FUNCTION_BLOCK Gerador_HMI (* HMI Gerador AGC150 - 74 vars + 33 HAB equipamentos *)
  (* Standard: 61499-2 *)
  (* Version 7.0, 13/05/2026, Claude *)
  PACKAGE Hidryco.HidrycoLib;
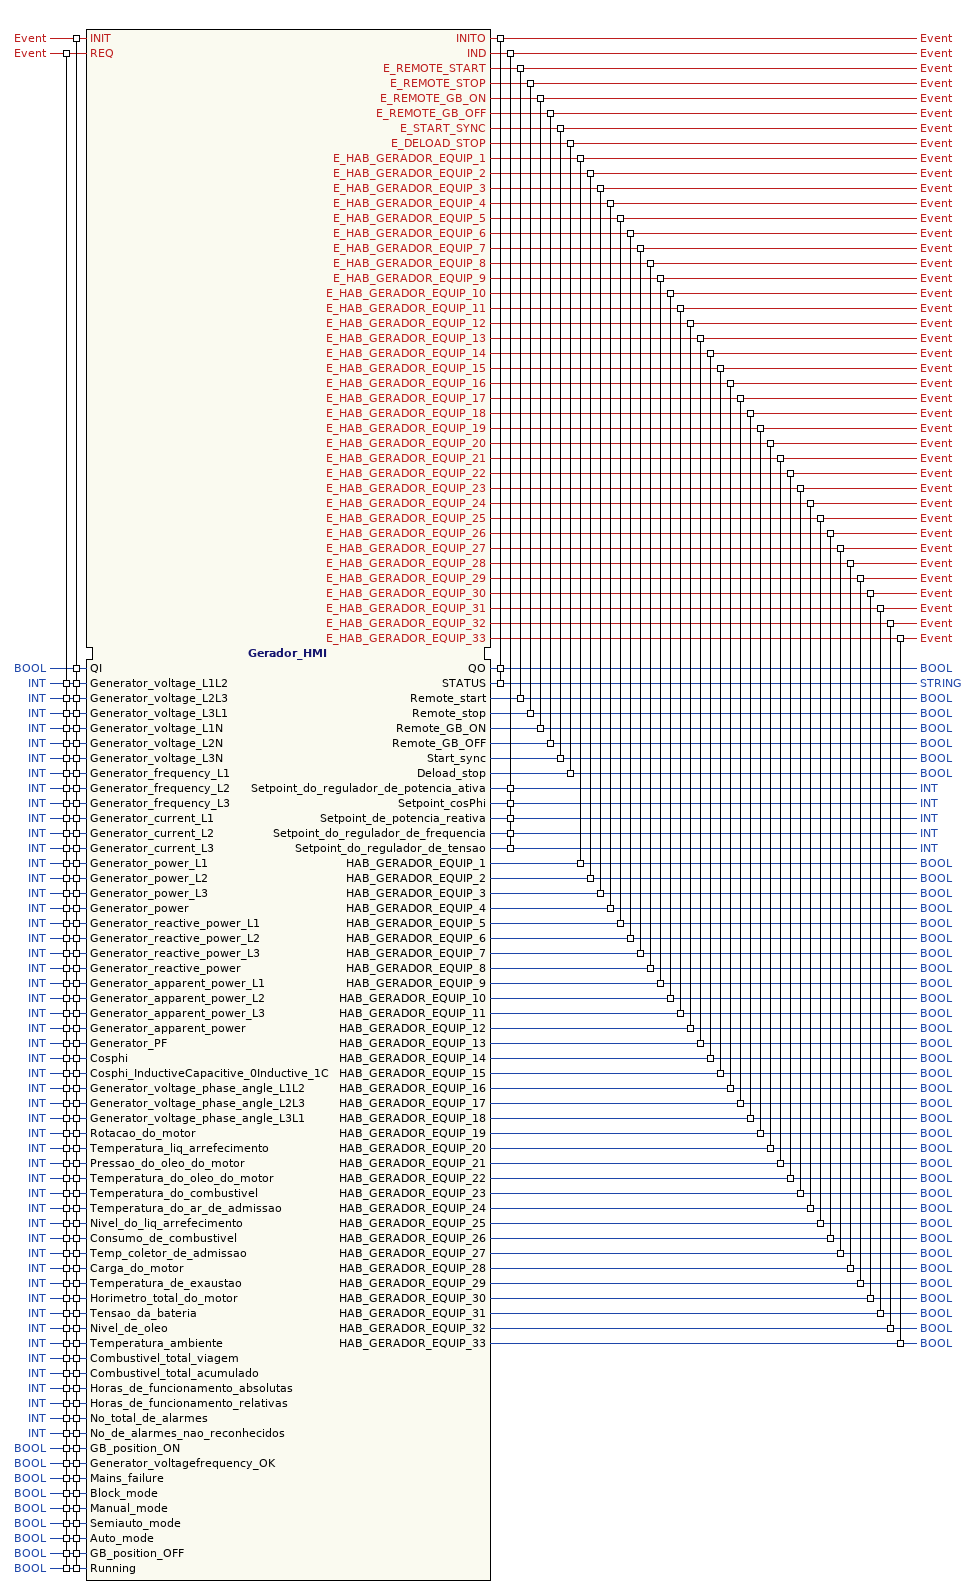
  EVENT_INPUT
    INIT WITH QI, Generator_voltage_L1L2, Generator_voltage_L2L3, Generator_voltage_L3L1, Generator_voltage_L1N, Generator_voltage_L2N, Generator_voltage_L3N, Generator_frequency_L1, Generator_frequency_L2, Generator_frequency_L3, Generator_current_L1, Generator_current_L2, Generator_current_L3, Generator_power_L1, Generator_power_L2, Generator_power_L3, Generator_power, Generator_reactive_power_L1, Generator_reactive_power_L2, Generator_reactive_power_L3, Generator_reactive_power, Generator_apparent_power_L1, Generator_apparent_power_L2, Generator_apparent_power_L3, Generator_apparent_power, Generator_PF, Cosphi, Cosphi_InductiveCapacitive_0Inductive_1C, Generator_voltage_phase_angle_L1L2, Generator_voltage_phase_angle_L2L3, Generator_voltage_phase_angle_L3L1, Rotacao_do_motor, Temperatura_liq_arrefecimento, Pressao_do_oleo_do_motor, Temperatura_do_oleo_do_motor, Temperatura_do_combustivel, Temperatura_do_ar_de_admissao, Nivel_do_liq_arrefecimento, Consumo_de_combustivel, Temp_coletor_de_admissao, Carga_do_motor, Temperatura_de_exaustao, Horimetro_total_do_motor, Tensao_da_bateria, Nivel_de_oleo, Temperatura_ambiente, Combustivel_total_viagem, Combustivel_total_acumulado, Horas_de_funcionamento_absolutas, Horas_de_funcionamento_relativas, No_total_de_alarmes, No_de_alarmes_nao_reconhecidos, GB_position_ON, Running, Generator_voltagefrequency_OK, Mains_failure, Block_mode, Manual_mode, Semiauto_mode, Auto_mode, GB_position_OFF;
    REQ WITH Generator_voltage_L1L2, Generator_voltage_L2L3, Generator_voltage_L3L1, Generator_voltage_L1N, Generator_voltage_L2N, Generator_voltage_L3N, Generator_frequency_L1, Generator_frequency_L2, Generator_frequency_L3, Generator_current_L1, Generator_current_L2, Generator_current_L3, Generator_power_L1, Generator_power_L2, Generator_power_L3, Generator_power, Generator_reactive_power_L1, Generator_reactive_power_L2, Generator_reactive_power_L3, Generator_reactive_power, Generator_apparent_power_L1, Generator_apparent_power_L2, Generator_apparent_power_L3, Generator_apparent_power, Generator_PF, Cosphi, Cosphi_InductiveCapacitive_0Inductive_1C, Generator_voltage_phase_angle_L1L2, Generator_voltage_phase_angle_L2L3, Generator_voltage_phase_angle_L3L1, Rotacao_do_motor, Temperatura_liq_arrefecimento, Pressao_do_oleo_do_motor, Temperatura_do_oleo_do_motor, Temperatura_do_combustivel, Temperatura_do_ar_de_admissao, Nivel_do_liq_arrefecimento, Consumo_de_combustivel, Temp_coletor_de_admissao, Carga_do_motor, Temperatura_de_exaustao, Horimetro_total_do_motor, Tensao_da_bateria, Nivel_de_oleo, Temperatura_ambiente, Combustivel_total_viagem, Combustivel_total_acumulado, Horas_de_funcionamento_absolutas, Horas_de_funcionamento_relativas, No_total_de_alarmes, No_de_alarmes_nao_reconhecidos, GB_position_ON, Running, Generator_voltagefrequency_OK, Mains_failure, Block_mode, Manual_mode, Semiauto_mode, Auto_mode, GB_position_OFF;
  END_EVENT
  EVENT_OUTPUT
    INITO WITH QO, STATUS;
    IND WITH Setpoint_do_regulador_de_potencia_ativa, Setpoint_cosPhi, Setpoint_de_potencia_reativa, Setpoint_do_regulador_de_frequencia, Setpoint_do_regulador_de_tensao;
    E_REMOTE_START WITH Remote_start;
    E_REMOTE_STOP WITH Remote_stop;
    E_REMOTE_GB_ON WITH Remote_GB_ON;
    E_REMOTE_GB_OFF WITH Remote_GB_OFF;
    E_START_SYNC WITH Start_sync;
    E_DELOAD_STOP WITH Deload_stop;
    E_HAB_GERADOR_EQUIP_1 WITH HAB_GERADOR_EQUIP_1;
    E_HAB_GERADOR_EQUIP_2 WITH HAB_GERADOR_EQUIP_2;
    E_HAB_GERADOR_EQUIP_3 WITH HAB_GERADOR_EQUIP_3;
    E_HAB_GERADOR_EQUIP_4 WITH HAB_GERADOR_EQUIP_4;
    E_HAB_GERADOR_EQUIP_5 WITH HAB_GERADOR_EQUIP_5;
    E_HAB_GERADOR_EQUIP_6 WITH HAB_GERADOR_EQUIP_6;
    E_HAB_GERADOR_EQUIP_7 WITH HAB_GERADOR_EQUIP_7;
    E_HAB_GERADOR_EQUIP_8 WITH HAB_GERADOR_EQUIP_8;
    E_HAB_GERADOR_EQUIP_9 WITH HAB_GERADOR_EQUIP_9;
    E_HAB_GERADOR_EQUIP_10 WITH HAB_GERADOR_EQUIP_10;
    E_HAB_GERADOR_EQUIP_11 WITH HAB_GERADOR_EQUIP_11;
    E_HAB_GERADOR_EQUIP_12 WITH HAB_GERADOR_EQUIP_12;
    E_HAB_GERADOR_EQUIP_13 WITH HAB_GERADOR_EQUIP_13;
    E_HAB_GERADOR_EQUIP_14 WITH HAB_GERADOR_EQUIP_14;
    E_HAB_GERADOR_EQUIP_15 WITH HAB_GERADOR_EQUIP_15;
    E_HAB_GERADOR_EQUIP_16 WITH HAB_GERADOR_EQUIP_16;
    E_HAB_GERADOR_EQUIP_17 WITH HAB_GERADOR_EQUIP_17;
    E_HAB_GERADOR_EQUIP_18 WITH HAB_GERADOR_EQUIP_18;
    E_HAB_GERADOR_EQUIP_19 WITH HAB_GERADOR_EQUIP_19;
    E_HAB_GERADOR_EQUIP_20 WITH HAB_GERADOR_EQUIP_20;
    E_HAB_GERADOR_EQUIP_21 WITH HAB_GERADOR_EQUIP_21;
    E_HAB_GERADOR_EQUIP_22 WITH HAB_GERADOR_EQUIP_22;
    E_HAB_GERADOR_EQUIP_23 WITH HAB_GERADOR_EQUIP_23;
    E_HAB_GERADOR_EQUIP_24 WITH HAB_GERADOR_EQUIP_24;
    E_HAB_GERADOR_EQUIP_25 WITH HAB_GERADOR_EQUIP_25;
    E_HAB_GERADOR_EQUIP_26 WITH HAB_GERADOR_EQUIP_26;
    E_HAB_GERADOR_EQUIP_27 WITH HAB_GERADOR_EQUIP_27;
    E_HAB_GERADOR_EQUIP_28 WITH HAB_GERADOR_EQUIP_28;
    E_HAB_GERADOR_EQUIP_29 WITH HAB_GERADOR_EQUIP_29;
    E_HAB_GERADOR_EQUIP_30 WITH HAB_GERADOR_EQUIP_30;
    E_HAB_GERADOR_EQUIP_31 WITH HAB_GERADOR_EQUIP_31;
    E_HAB_GERADOR_EQUIP_32 WITH HAB_GERADOR_EQUIP_32;
    E_HAB_GERADOR_EQUIP_33 WITH HAB_GERADOR_EQUIP_33;
  END_EVENT
  VAR_INPUT
    QI : BOOL;
    Generator_voltage_L1L2 : INT; (* Generator voltage L1L2 *)
    Generator_voltage_L2L3 : INT; (* Generator voltage L2L3 *)
    Generator_voltage_L3L1 : INT; (* Generator voltage L3L1 *)
    Generator_voltage_L1N : INT; (* Generator voltage L1N *)
    Generator_voltage_L2N : INT; (* Generator voltage L2N *)
    Generator_voltage_L3N : INT; (* Generator voltage L3N *)
    Generator_frequency_L1 : INT; (* Generator frequency L1 *)
    Generator_frequency_L2 : INT; (* Generator frequency L2 *)
    Generator_frequency_L3 : INT; (* Generator frequency L3 *)
    Generator_current_L1 : INT; (* Generator current L1 *)
    Generator_current_L2 : INT; (* Generator current L2 *)
    Generator_current_L3 : INT; (* Generator current L3 *)
    Generator_power_L1 : INT; (* Generator power L1 *)
    Generator_power_L2 : INT; (* Generator power L2 *)
    Generator_power_L3 : INT; (* Generator power L3 *)
    Generator_power : INT; (* Generator power *)
    Generator_reactive_power_L1 : INT; (* Generator reactive power L1 *)
    Generator_reactive_power_L2 : INT; (* Generator reactive power L2 *)
    Generator_reactive_power_L3 : INT; (* Generator reactive power L3 *)
    Generator_reactive_power : INT; (* Generator reactive power *)
    Generator_apparent_power_L1 : INT; (* Generator apparent power L1 *)
    Generator_apparent_power_L2 : INT; (* Generator apparent power L2 *)
    Generator_apparent_power_L3 : INT; (* Generator apparent power L3 *)
    Generator_apparent_power : INT; (* Generator apparent power *)
    Generator_PF : INT; (* Generator PF *)
    Cosphi : INT; (* Cosphi *)
    Cosphi_InductiveCapacitive_0Inductive_1C : INT; (* Cosphi InductiveCapacitive 0Inductive 1C *)
    Generator_voltage_phase_angle_L1L2 : INT; (* Generator voltage phase angle L1L2 *)
    Generator_voltage_phase_angle_L2L3 : INT; (* Generator voltage phase angle L2L3 *)
    Generator_voltage_phase_angle_L3L1 : INT; (* Generator voltage phase angle L3L1 *)
    Rotacao_do_motor : INT; (* Rotacao do motor *)
    Temperatura_liq_arrefecimento : INT; (* Temperatura liq arrefecimento *)
    Pressao_do_oleo_do_motor : INT; (* Pressao do oleo do motor *)
    Temperatura_do_oleo_do_motor : INT; (* Temperatura do oleo do motor *)
    Temperatura_do_combustivel : INT; (* Temperatura do combustivel *)
    Temperatura_do_ar_de_admissao : INT; (* Temperatura do ar de admissao *)
    Nivel_do_liq_arrefecimento : INT; (* Nivel do liq arrefecimento *)
    Consumo_de_combustivel : INT; (* Consumo de combustivel *)
    Temp_coletor_de_admissao : INT; (* Temp coletor de admissao *)
    Carga_do_motor : INT; (* Carga do motor *)
    Temperatura_de_exaustao : INT; (* Temperatura de exaustao *)
    Horimetro_total_do_motor : INT; (* Horimetro total do motor *)
    Tensao_da_bateria : INT; (* Tensao da bateria *)
    Nivel_de_oleo : INT; (* Nivel de oleo *)
    Temperatura_ambiente : INT; (* Temperatura ambiente *)
    Combustivel_total_viagem : INT; (* Combustivel total viagem *)
    Combustivel_total_acumulado : INT; (* Combustivel total acumulado *)
    Horas_de_funcionamento_absolutas : INT; (* Horas de funcionamento absolutas *)
    Horas_de_funcionamento_relativas : INT; (* Horas de funcionamento relativas *)
    No_total_de_alarmes : INT; (* No total de alarmes *)
    No_de_alarmes_nao_reconhecidos : INT; (* No de alarmes nao reconhecidos *)
    GB_position_ON : BOOL; (* GB position ON *)
    Generator_voltagefrequency_OK : BOOL; (* Generator voltagefrequency OK *)
    Mains_failure : BOOL; (* Mains failure *)
    Block_mode : BOOL; (* Block mode *)
    Manual_mode : BOOL; (* Manual mode *)
    Semiauto_mode : BOOL; (* Semiauto mode *)
    Auto_mode : BOOL; (* Auto mode *)
    GB_position_OFF : BOOL; (* GB position OFF *)
    Running : BOOL; (* Running *)
  END_VAR
  VAR_OUTPUT
    QO : BOOL;
    STATUS : STRING;
    Remote_start : BOOL; (* Remote start *)
    Remote_stop : BOOL; (* Remote stop *)
    Remote_GB_ON : BOOL; (* Remote GB ON *)
    Remote_GB_OFF : BOOL; (* Remote GB OFF *)
    Start_sync : BOOL; (* Start sync *)
    Deload_stop : BOOL; (* Deload stop *)
    Setpoint_do_regulador_de_potencia_ativa : INT; (* Setpoint do regulador de potencia ativa *)
    Setpoint_cosPhi : INT; (* Setpoint cosPhi *)
    Setpoint_de_potencia_reativa : INT; (* Setpoint de potencia reativa *)
    Setpoint_do_regulador_de_frequencia : INT; (* Setpoint do regulador de frequencia *)
    Setpoint_do_regulador_de_tensao : INT; (* Setpoint do regulador de tensao *)
    HAB_GERADOR_EQUIP_1 : BOOL; (* Habilitar equipamento 1 no gerador *)
    HAB_GERADOR_EQUIP_2 : BOOL; (* Habilitar equipamento 2 no gerador *)
    HAB_GERADOR_EQUIP_3 : BOOL; (* Habilitar equipamento 3 no gerador *)
    HAB_GERADOR_EQUIP_4 : BOOL; (* Habilitar equipamento 4 no gerador *)
    HAB_GERADOR_EQUIP_5 : BOOL; (* Habilitar equipamento 5 no gerador *)
    HAB_GERADOR_EQUIP_6 : BOOL; (* Habilitar equipamento 6 no gerador *)
    HAB_GERADOR_EQUIP_7 : BOOL; (* Habilitar equipamento 7 no gerador *)
    HAB_GERADOR_EQUIP_8 : BOOL; (* Habilitar equipamento 8 no gerador *)
    HAB_GERADOR_EQUIP_9 : BOOL; (* Habilitar equipamento 9 no gerador *)
    HAB_GERADOR_EQUIP_10 : BOOL; (* Habilitar equipamento 10 no gerador *)
    HAB_GERADOR_EQUIP_11 : BOOL; (* Habilitar equipamento 11 no gerador *)
    HAB_GERADOR_EQUIP_12 : BOOL; (* Habilitar equipamento 12 no gerador *)
    HAB_GERADOR_EQUIP_13 : BOOL; (* Habilitar equipamento 13 no gerador *)
    HAB_GERADOR_EQUIP_14 : BOOL; (* Habilitar equipamento 14 no gerador *)
    HAB_GERADOR_EQUIP_15 : BOOL; (* Habilitar equipamento 15 no gerador *)
    HAB_GERADOR_EQUIP_16 : BOOL; (* Habilitar equipamento 16 no gerador *)
    HAB_GERADOR_EQUIP_17 : BOOL; (* Habilitar equipamento 17 no gerador *)
    HAB_GERADOR_EQUIP_18 : BOOL; (* Habilitar equipamento 18 no gerador *)
    HAB_GERADOR_EQUIP_19 : BOOL; (* Habilitar equipamento 19 no gerador *)
    HAB_GERADOR_EQUIP_20 : BOOL; (* Habilitar equipamento 20 no gerador *)
    HAB_GERADOR_EQUIP_21 : BOOL; (* Habilitar equipamento 21 no gerador *)
    HAB_GERADOR_EQUIP_22 : BOOL; (* Habilitar equipamento 22 no gerador *)
    HAB_GERADOR_EQUIP_23 : BOOL; (* Habilitar equipamento 23 no gerador *)
    HAB_GERADOR_EQUIP_24 : BOOL; (* Habilitar equipamento 24 no gerador *)
    HAB_GERADOR_EQUIP_25 : BOOL; (* Habilitar equipamento 25 no gerador *)
    HAB_GERADOR_EQUIP_26 : BOOL; (* Habilitar equipamento 26 no gerador *)
    HAB_GERADOR_EQUIP_27 : BOOL; (* Habilitar equipamento 27 no gerador *)
    HAB_GERADOR_EQUIP_28 : BOOL; (* Habilitar equipamento 28 no gerador *)
    HAB_GERADOR_EQUIP_29 : BOOL; (* Habilitar equipamento 29 no gerador *)
    HAB_GERADOR_EQUIP_30 : BOOL; (* Habilitar equipamento 30 no gerador *)
    HAB_GERADOR_EQUIP_31 : BOOL; (* Habilitar equipamento 31 no gerador *)
    HAB_GERADOR_EQUIP_32 : BOOL; (* Habilitar equipamento 32 no gerador *)
    HAB_GERADOR_EQUIP_33 : BOOL; (* Habilitar equipamento 33 no gerador *)
  END_VAR
  SERVICE /
    SEQUENCE 
    END_SEQUENCE
  END_SERVICE
END_FUNCTION_BLOCK
